INTERFACE ITF_EM_Template EXTENDS ITF_EM_Base

{attribute 'monitoring' := 'call'}
PROPERTY p_rstConfig : REFERENCE TO ST_EM_Template_Config
GET
END_GET
END_PROPERTY

END_INTERFACE

(* stored: Version 1.1.0.1, ProductVersion 3.1.4024.10
   Itf ITF_EM_Template: Id {6c2104cf-2e12-4fb5-af04-a804f5784aaa}
   Property p_rstConfig: Id {fce17ab7-6700-41e2-8106-c8a60c202f59}
   Get Get: Id {d43d2520-6ed8-453b-b49f-75115fc828f6} *)
